// TIA Portal V20 export
VAR_GLOBAL   // PLC tag table "Unit1Em0_Servo"
END_VAR
